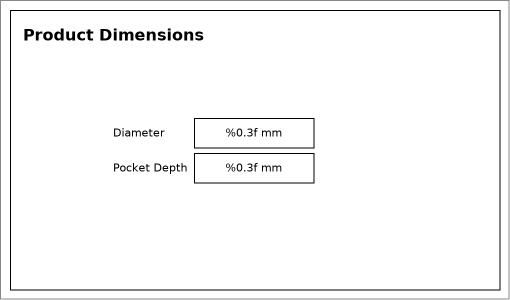
VISUALIZATION Settings_ProductDimensions  // 510x300
VAR_IN_OUT
	Diameter	: LREAL;
	PocketDepth	: LREAL;
END_VAR
    Rectangle (10,10 490x280)
    Group (110,118 204x65)
        Label (0,0 60x30), "Diameter"
        Rectangle (84,0 120x30), "%0.3f mm", text variable: Diameter
            OnMouseClick: write Diameter via Default
        Rectangle (84,35 120x30), "%0.3f mm", text variable: PocketDepth
            OnMouseClick: write PocketDepth via Default
        Label (0,35 80x30), "Pocket Depth"
    Label (20,20 150x30), "Product Dimensions"
END_VISUALIZATION

(* stored: Version 1.1.0.1, ProductVersion 3.1.4024.3
   Visu Settings_ProductDimensions: Id {995f8b03-856a-4a7a-be91-7d184c5baed1} *)
